(* Logix 5000 project; controller Traffic_light_test vendor 1 type 14 code 54 rev 20.11; software revision 20.05 *)

TASK MainTask (continuous, watchdog 500 ms) : MainProgram

MODULES
   Local : vendor 1 type 14 code 54 (ICP 0, rev 20.11)
       : 1756-IA16 (ICP 8, rev 2.1, Input RPI 20 ms)
       : 1756-OW16I (ICP 9, rev 1.1, Output RPI 20 ms)
END_MODULES

PROGRAM MainProgram   (* main routine MainRoutine *)
VAR
   CTU1 : COUNTER := (PRE := 10, ACC := 1);
   CTU2 : COUNTER := (PRE := 10, ACC := 1);
   CTU3 : COUNTER := (PRE := 10, ACC := 1);
   CTU4 : COUNTER := (PRE := 10, ACC := 1);
   Green1 : ALIAS FOR Local:9:O.Data.0;
   Green2 : ALIAS FOR Local:9:O.Data.1;
   Green3 : ALIAS FOR Local:9:O.Data.2;
   Green4 : ALIAS FOR Local:9:O.Data.3;
   Green_Timer1 : TIMER := (PRE := 16000);
   Green_Timer2 : TIMER := (PRE := 20000);
   Green_Timer21 : TIMER := (PRE := 16000);
   Green_Timer22 : TIMER := (PRE := 20000);
   Green_Timer23 : TIMER := (PRE := 22000);
   Green_Timer24 : TIMER := (PRE := 26000);
   Green_Timer3 : TIMER := (PRE := 22000);
   Green_timer31 : TIMER := (PRE := 16000);
   Green_timer32 : TIMER := (PRE := 20000);
   Green_timer33 : TIMER := (PRE := 24000);
   Green_timer34 : TIMER := (PRE := 26000);
   Green_Timer4 : TIMER := (PRE := 26000);
   Green_timer41 : TIMER := (PRE := 16000);
   Green_timer42 : TIMER := (PRE := 18000);
   Green_timer43 : TIMER := (PRE := 23000);
   Green_timer44 : TIMER := (PRE := 26000);
   Red1 : ALIAS FOR Local:9:O.Data.4;
   Red2 : ALIAS FOR Local:9:O.Data.7;
   Red3 : ALIAS FOR Local:9:O.Data.5;
   Red4 : ALIAS FOR Local:9:O.Data.6;
END_VAR

ROUTINE High_traffic1   (* ladder *)
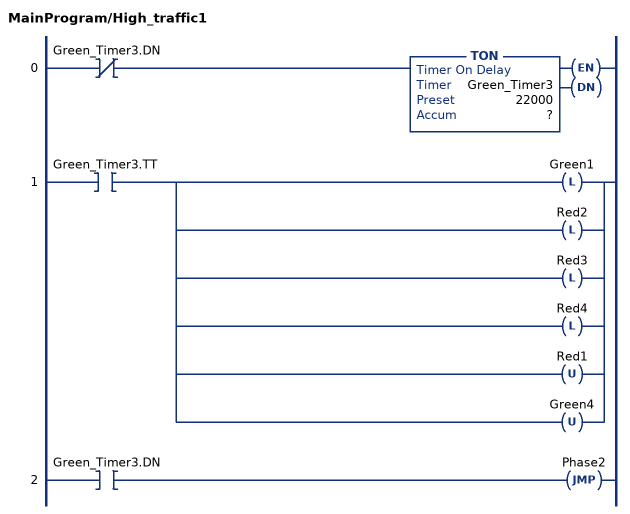
   0: XIO(Green_Timer3.DN)TON(Green_Timer3,?,?);
   1: XIC(Green_Timer3.TT)[OTL(Green1) ,OTL(Red2) ,OTL(Red3) ,OTL(Red4) ,OTU(Red1) ,OTU(Green4) ];
   2: XIC(Green_Timer3.DN)JMP(Phase2);
END_ROUTINE

ROUTINE High_traffic2   (* ladder *)
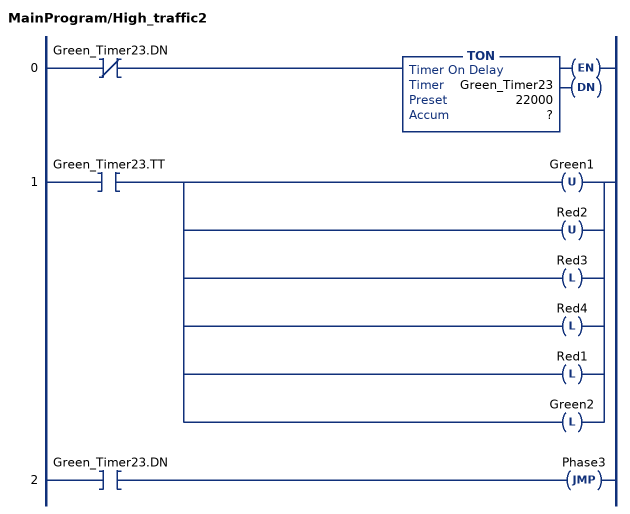
   0: XIO(Green_Timer23.DN)TON(Green_Timer23,?,?);
   1: XIC(Green_Timer23.TT)[OTU(Green1) ,OTU(Red2) ,OTL(Red3) ,OTL(Red4) ,OTL(Red1) ,OTL(Green2) ];
   2: XIC(Green_Timer23.DN)JMP(Phase3);
END_ROUTINE

ROUTINE High_traffic3   (* ladder *)
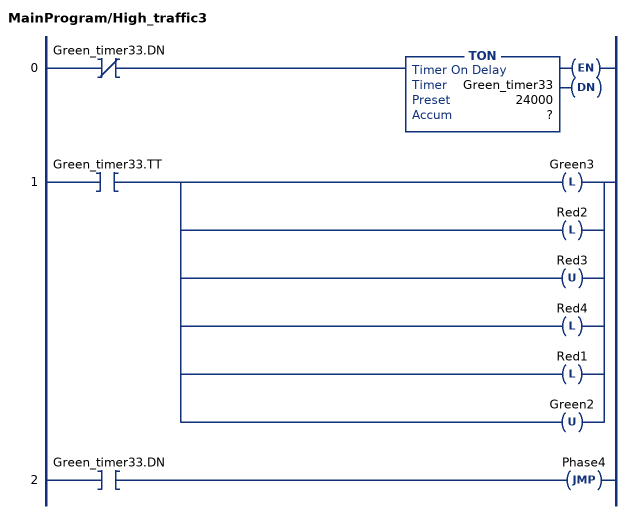
   0: XIO(Green_timer33.DN)TON(Green_timer33,?,?);
   1: XIC(Green_timer33.TT)[OTL(Green3) ,OTL(Red2) ,OTU(Red3) ,OTL(Red4) ,OTL(Red1) ,OTU(Green2) ];
   2: XIC(Green_timer33.DN)JMP(Phase4);
END_ROUTINE

ROUTINE High_traffic4   (* ladder *)
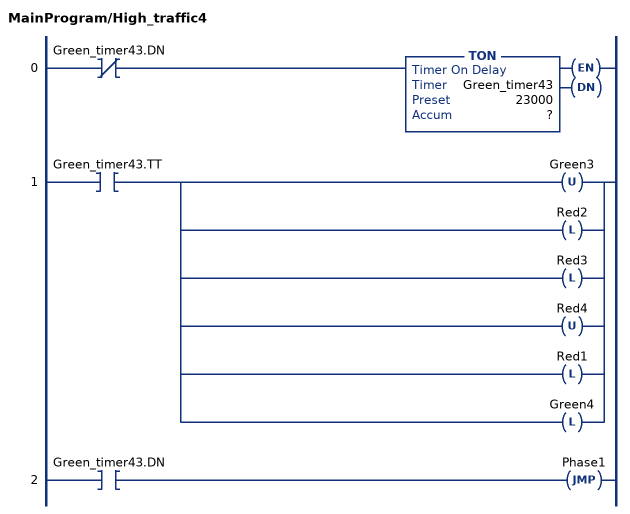
   0: XIO(Green_timer43.DN)TON(Green_timer43,?,?);
   1: XIC(Green_timer43.TT)[OTU(Green3) ,OTL(Red2) ,OTL(Red3) ,OTU(Red4) ,OTL(Red1) ,OTL(Green4) ];
   2: XIC(Green_timer43.DN)JMP(Phase1);
END_ROUTINE

ROUTINE Low_traffic1   (* ladder *)
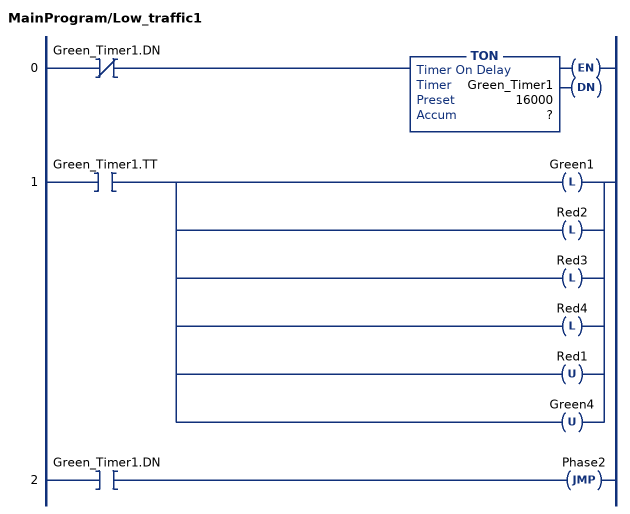
   0: XIO(Green_Timer1.DN)TON(Green_Timer1,?,?);
   1: XIC(Green_Timer1.TT)[OTL(Green1) ,OTL(Red2) ,OTL(Red3) ,OTL(Red4) ,OTU(Red1) ,OTU(Green4) ];
   2: XIC(Green_Timer1.DN)JMP(Phase2);
END_ROUTINE

ROUTINE Low_traffic2   (* ladder *)
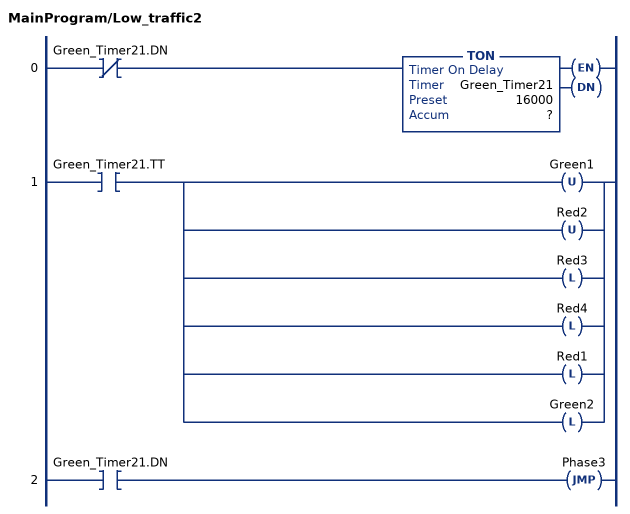
   0: XIO(Green_Timer21.DN)TON(Green_Timer21,?,?);
   1: XIC(Green_Timer21.TT)[OTU(Green1) ,OTU(Red2) ,OTL(Red3) ,OTL(Red4) ,OTL(Red1) ,OTL(Green2) ];
   2: XIC(Green_Timer21.DN)JMP(Phase3);
END_ROUTINE

ROUTINE Low_traffic3   (* ladder *)
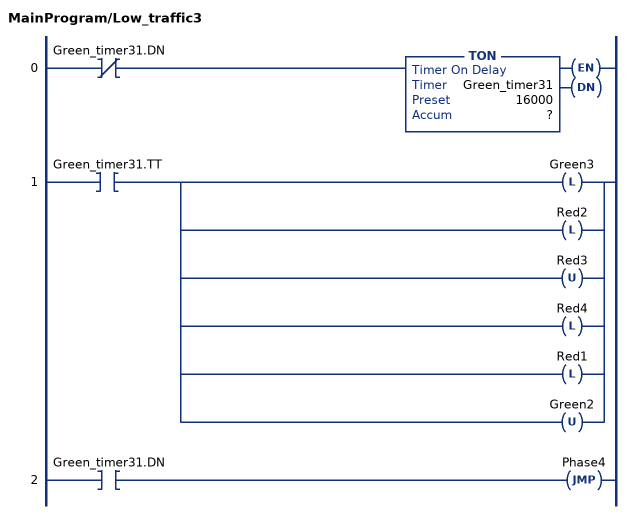
   0: XIO(Green_timer31.DN)TON(Green_timer31,?,?);
   1: XIC(Green_timer31.TT)[OTL(Green3) ,OTL(Red2) ,OTU(Red3) ,OTL(Red4) ,OTL(Red1) ,OTU(Green2) ];
   2: XIC(Green_timer31.DN)JMP(Phase4);
END_ROUTINE

ROUTINE Low_traffic4   (* ladder *)
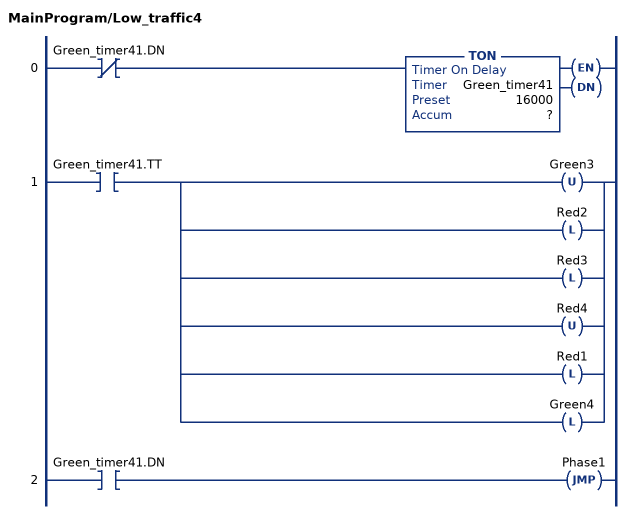
   0: XIO(Green_timer41.DN)TON(Green_timer41,?,?);
   1: XIC(Green_timer41.TT)[OTU(Green3) ,OTL(Red2) ,OTL(Red3) ,OTU(Red4) ,OTL(Red1) ,OTL(Green4) ];
   2: XIC(Green_timer41.DN)JMP(Phase1);
END_ROUTINE

ROUTINE MainRoutine   (* ladder *)
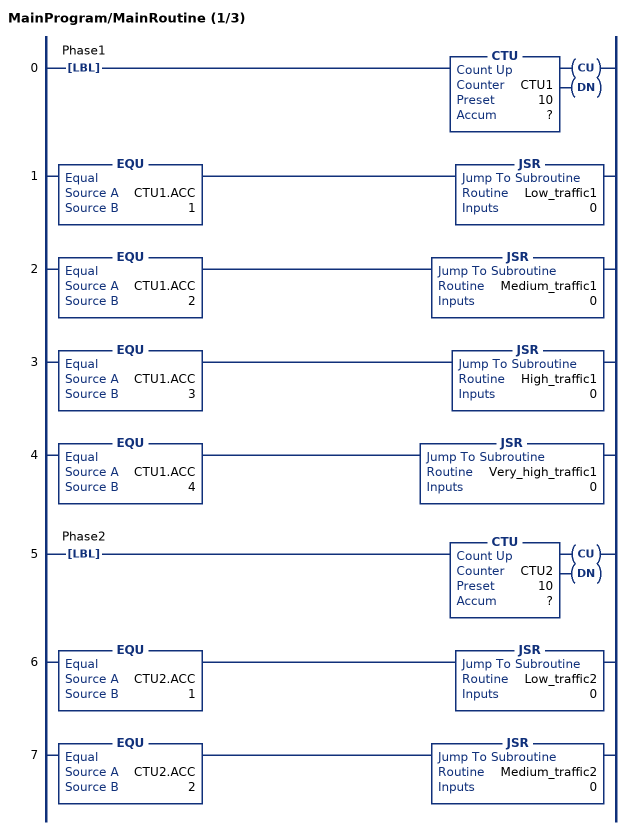
   0: LBL(Phase1)CTU(CTU1,?,?);
   1: EQU(CTU1.ACC,1)JSR(Low_traffic1,0);
   2: EQU(CTU1.ACC,2)JSR(Medium_traffic1,0);
   3: EQU(CTU1.ACC,3)JSR(High_traffic1,0);
   4: EQU(CTU1.ACC,4)JSR(Very_high_traffic1,0);
   5: LBL(Phase2)CTU(CTU2,?,?);
   6: EQU(CTU2.ACC,1)JSR(Low_traffic2,0);
   7: EQU(CTU2.ACC,2)JSR(Medium_traffic2,0);
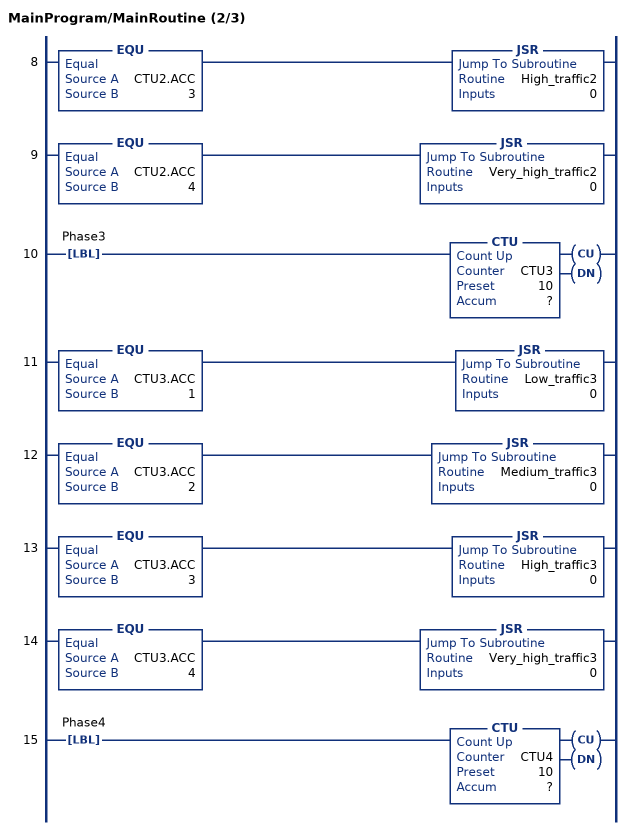
   8: EQU(CTU2.ACC,3)JSR(High_traffic2,0);
   9: EQU(CTU2.ACC,4)JSR(Very_high_traffic2,0);
   10: LBL(Phase3)CTU(CTU3,?,?);
   11: EQU(CTU3.ACC,1)JSR(Low_traffic3,0);
   12: EQU(CTU3.ACC,2)JSR(Medium_traffic3,0);
   13: EQU(CTU3.ACC,3)JSR(High_traffic3,0);
   14: EQU(CTU3.ACC,4)JSR(Very_high_traffic3,0);
   15: LBL(Phase4)CTU(CTU4,?,?);
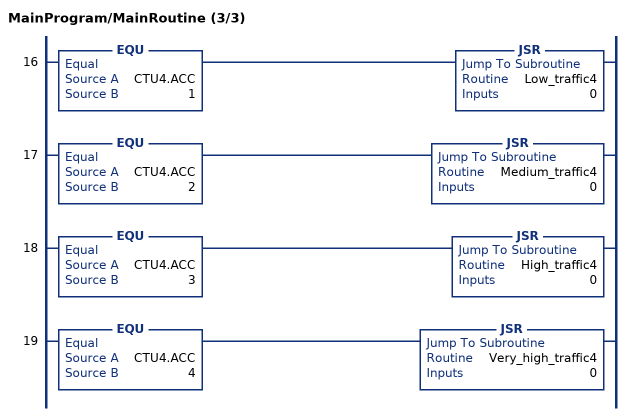
   16: EQU(CTU4.ACC,1)JSR(Low_traffic4,0);
   17: EQU(CTU4.ACC,2)JSR(Medium_traffic4,0);
   18: EQU(CTU4.ACC,3)JSR(High_traffic4,0);
   19: EQU(CTU4.ACC,4)JSR(Very_high_traffic4,0);
END_ROUTINE

ROUTINE Medium_traffic1   (* ladder *)
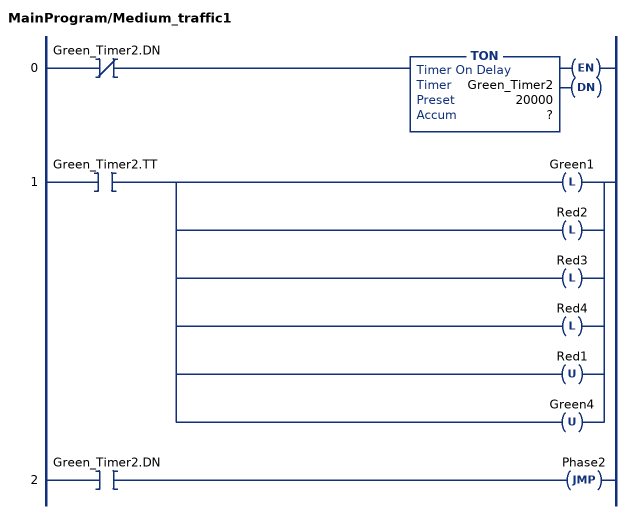
   0: XIO(Green_Timer2.DN)TON(Green_Timer2,?,?);
   1: XIC(Green_Timer2.TT)[OTL(Green1) ,OTL(Red2) ,OTL(Red3) ,OTL(Red4) ,OTU(Red1) ,OTU(Green4) ];
   2: XIC(Green_Timer2.DN)JMP(Phase2);
END_ROUTINE

ROUTINE Medium_traffic2   (* ladder *)
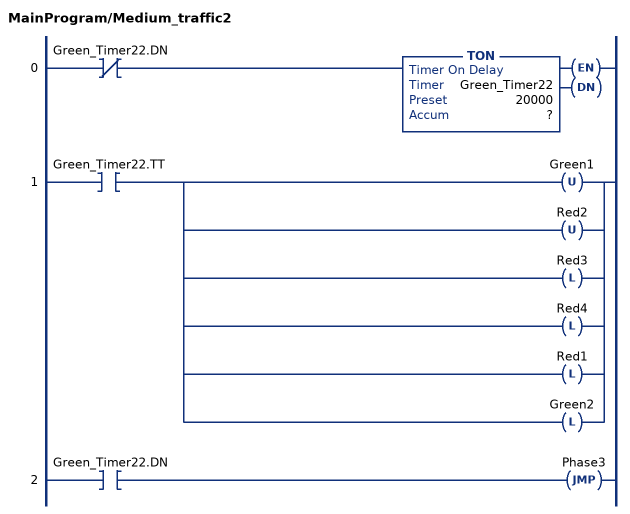
   0: XIO(Green_Timer22.DN)TON(Green_Timer22,?,?);
   1: XIC(Green_Timer22.TT)[OTU(Green1) ,OTU(Red2) ,OTL(Red3) ,OTL(Red4) ,OTL(Red1) ,OTL(Green2) ];
   2: XIC(Green_Timer22.DN)JMP(Phase3);
END_ROUTINE

ROUTINE Medium_traffic3   (* ladder *)
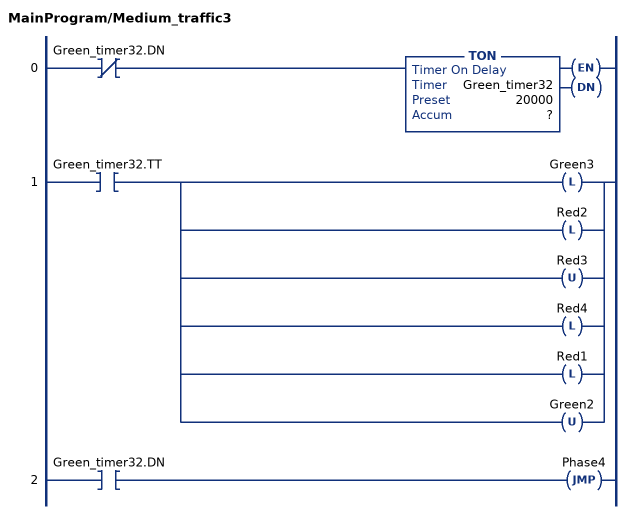
   0: XIO(Green_timer32.DN)TON(Green_timer32,?,?);
   1: XIC(Green_timer32.TT)[OTL(Green3) ,OTL(Red2) ,OTU(Red3) ,OTL(Red4) ,OTL(Red1) ,OTU(Green2) ];
   2: XIC(Green_timer32.DN)JMP(Phase4);
END_ROUTINE

ROUTINE Medium_traffic4   (* ladder *)
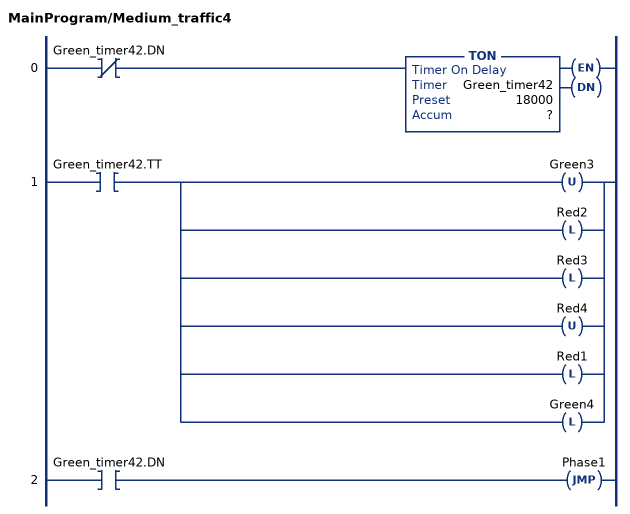
   0: XIO(Green_timer42.DN)TON(Green_timer42,?,?);
   1: XIC(Green_timer42.TT)[OTU(Green3) ,OTL(Red2) ,OTL(Red3) ,OTU(Red4) ,OTL(Red1) ,OTL(Green4) ];
   2: XIC(Green_timer42.DN)JMP(Phase1);
END_ROUTINE

ROUTINE Very_high_traffic1   (* ladder *)
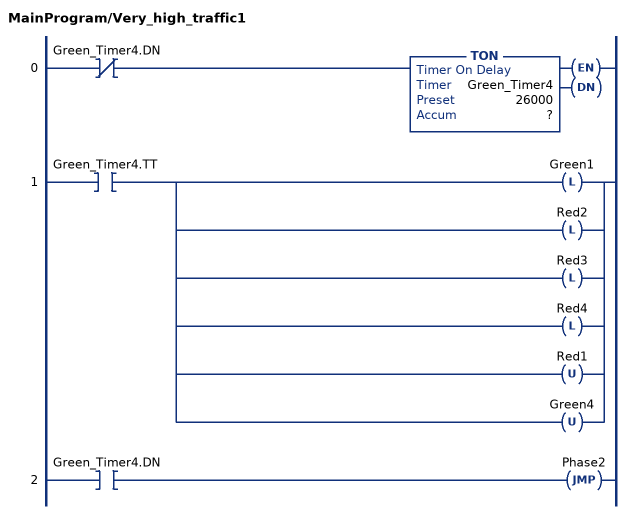
   0: XIO(Green_Timer4.DN)TON(Green_Timer4,?,?);
   1: XIC(Green_Timer4.TT)[OTL(Green1) ,OTL(Red2) ,OTL(Red3) ,OTL(Red4) ,OTU(Red1) ,OTU(Green4) ];
   2: XIC(Green_Timer4.DN)JMP(Phase2);
END_ROUTINE

ROUTINE Very_high_traffic2   (* ladder *)
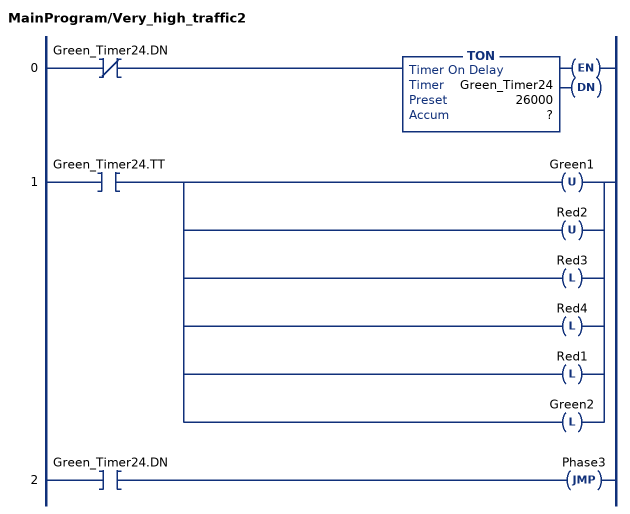
   0: XIO(Green_Timer24.DN)TON(Green_Timer24,?,?);
   1: XIC(Green_Timer24.TT)[OTU(Green1) ,OTU(Red2) ,OTL(Red3) ,OTL(Red4) ,OTL(Red1) ,OTL(Green2) ];
   2: XIC(Green_Timer24.DN)JMP(Phase3);
END_ROUTINE

ROUTINE Very_high_traffic3   (* ladder *)
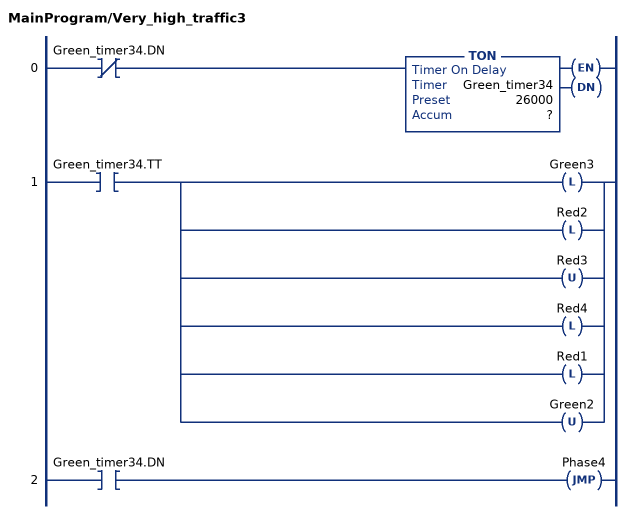
   0: XIO(Green_timer34.DN)TON(Green_timer34,?,?);
   1: XIC(Green_timer34.TT)[OTL(Green3) ,OTL(Red2) ,OTU(Red3) ,OTL(Red4) ,OTL(Red1) ,OTU(Green2) ];
   2: XIC(Green_timer34.DN)JMP(Phase4);
END_ROUTINE

ROUTINE Very_high_traffic4   (* ladder *)
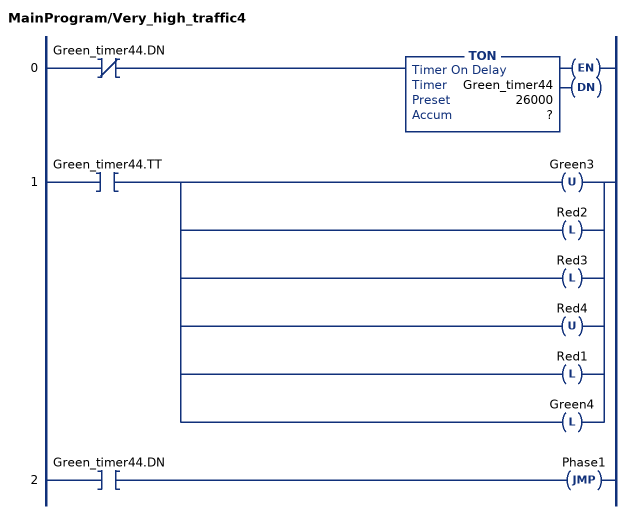
   0: XIO(Green_timer44.DN)TON(Green_timer44,?,?);
   1: XIC(Green_timer44.TT)[OTU(Green3) ,OTL(Red2) ,OTL(Red3) ,OTU(Red4) ,OTL(Red1) ,OTL(Green4) ];
   2: XIC(Green_timer44.DN)JMP(Phase1);
END_ROUTINE
END_PROGRAM
